// TIA Portal V20 export
TYPE "LER_typeGearInCommand"
// stored: Access Published
   STRUCT
      execute : Bool;
      continuousUpdate : Bool;
      ratioNumerator : DInt;
      ratioDenominator : DInt;
      acceleration : LReal;
      deceleration : LReal;
      jerk : LReal;
      positionControlled : Bool;
   END_STRUCT;
END_TYPE
